FUNCTION_BLOCK "Syntax_ForMissingDo"
{ S7_Optimized_Access := 'TRUE' }
VERSION : 0.1

VAR
    a        : Int := 1;
    b        : Int := 2;
    result   : Int := 0;
    flag     : Bool := TRUE;
    i        : Int := 0;
    values   : Array[0..9] of Int;
END_VAR
BEGIN
    FOR #i := 0 TO 9
        #values[#i] := #i;
    END_FOR;
    // EXPECT: error[syntax.for-missing-do] SYN-FOR-003

END_FUNCTION_BLOCK
